Fanuc KAREL source: kt00441.KL

-- PROVISIONAL review KL for V1013-1; original PC SHA256 4e34bf3060be322d8ce4038728e2d5165975f9ca4947b02bff871571ce28ceae
-- Incomplete behavior may be omitted. Consult companion uncertainty JSON. Do not deploy.
PROGRAM KT00441
%NOLOCKGROUP
VAR
  R1 : REAL
  I2 : INTEGER
  OUT : BOOLEAN
BEGIN
  -- UNRESOLVED_PC offsets 5-16; opcodes 2E,23
  -- UNRESOLVED_PC offsets 21-32; opcodes 2E,23
  -- UNRESOLVED_PC offsets 37-57; opcodes 21,21,64,72,23
  -- UNRESOLVED_PC offsets 62-66; opcodes 7F
END KT00441
